(* IEC 61131-3 sources: CannyIEC/st/library_information, 1 file *)

(* ---- getlibversion-GetLibVersion.st ---- *)
(* --- Interface --- *)
// This function has been automatically generated from the project information.
FUNCTION GetLibVersion : VERSION
VAR_INPUT

END_VAR
(* --- Implementation --- *)
GetLibVersion.uiMajor := 0;
GetLibVersion.uiMinor := 3;
GetLibVersion.uiServicePack := 19;
GetLibVersion.uiPatch := 15;
